PROGRAM F13_CaseContentValidation_ORG
VAR
	fbCrossPushCounter					: CTU;
	bCaseCompleteInsidePacker			: BOOL;


	rtrigSetEarlyCaseValidationOK			: R_TRIG;
	rtrigSetEarlyCaseValidationNOK		: R_TRIG;

	fbBiuldPackerLogString				: FB_CASE_BiuldPackerLogString;
	fbShiftPackerQueue					: FB_CASE_ShiftPackerQueue;
	fbMovePackerToCase				: FB_CASE_MovePackerToCase;
	fbFinaliseCaseData					: FB_CASE_FinaliseCaseData;

	fbValidationIndexOK					: FB_CTU32;
	fbValidationIndexNoData				: FB_CTU32;
	fbValidationIndexUnder				: FB_CTU32;
	fbValidationIndexOver				: FB_CTU32;


	fbDebugCNT				: FB_DEBUG_CounterArray;
	aCNTDebug				: ARRAY [1..10] OF UDINT;
	bResetCNT					: BOOL;


END_VAR

(*
Modification history:
Date		|	Author 		|	Remark
----------------------------------------------------------------------------------------------------
02.09.20	|	PP			|	Start Remarking.
*)

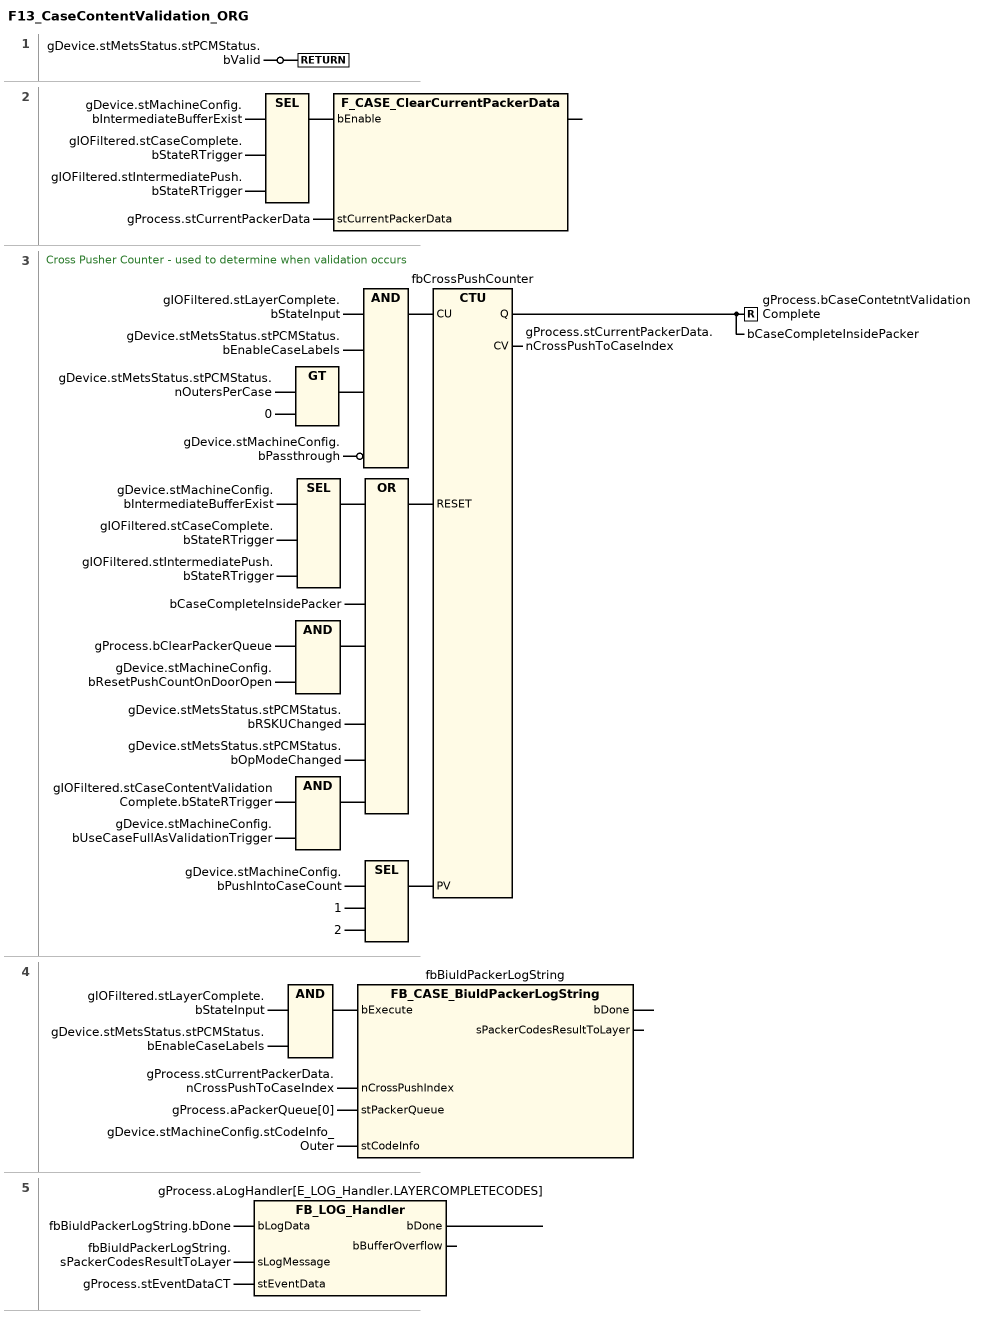
// NETWORK 1
IF NOT gDevice.stMetsStatus.stPCMStatus.bValid THEN RETURN; END_IF

// NETWORK 2
F_CASE_ClearCurrentPackerData(bEnable := SEL(gDevice.stMachineConfig.bIntermediateBufferExist, gIOFiltered.stCaseComplete.bStateRTrigger, gIOFiltered.stIntermediatePush.bStateRTrigger), stCurrentPackerData := gProcess.stCurrentPackerData);

// NETWORK 3
// 					Cross Pusher Counter - used to determine when validation occurs
//
//
fbCrossPushCounter(
    CU := gIOFiltered.stLayerComplete.bStateInput AND gDevice.stMetsStatus.stPCMStatus.bEnableCaseLabels AND gDevice.stMetsStatus.stPCMStatus.nOutersPerCase > 0 AND NOT gDevice.stMachineConfig.bPassthrough,
    RESET := SEL(gDevice.stMachineConfig.bIntermediateBufferExist, gIOFiltered.stCaseComplete.bStateRTrigger, gIOFiltered.stIntermediatePush.bStateRTrigger) OR bCaseCompleteInsidePacker OR gProcess.bClearPackerQueue AND gDevice.stMachineConfig.bResetPushCountOnDoorOpen OR gDevice.stMetsStatus.stPCMStatus.bRSKUChanged OR gDevice.stMetsStatus.stPCMStatus.bOpModeChanged OR gIOFiltered.stCaseContentValidationComplete.bStateRTrigger AND gDevice.stMachineConfig.bUseCaseFullAsValidationTrigger,
    PV := SEL(gDevice.stMachineConfig.bPushIntoCaseCount, 1, 2),
    CV => gProcess.stCurrentPackerData.nCrossPushToCaseIndex); // CTU
gProcess.bCaseContetntValidationComplete R= fbCrossPushCounter.Q;
bCaseCompleteInsidePacker := fbCrossPushCounter.Q;

// NETWORK 4
fbBiuldPackerLogString(
    bExecute := gIOFiltered.stLayerComplete.bStateInput AND gDevice.stMetsStatus.stPCMStatus.bEnableCaseLabels,
    nCrossPushIndex := gProcess.stCurrentPackerData.nCrossPushToCaseIndex,
    stPackerQueue := gProcess.aPackerQueue[0],
    stCodeInfo := gDevice.stMachineConfig.stCodeInfo_Outer); // FB_CASE_BiuldPackerLogString

// NETWORK 5
gProcess.aLogHandler[E_LOG_Handler.LAYERCOMPLETECODES](
    bLogData := fbBiuldPackerLogString.bDone,
    sLogMessage := fbBiuldPackerLogString.sPackerCodesResultToLayer,
    stEventData := gProcess.stEventDataCT); // FB_LOG_Handler

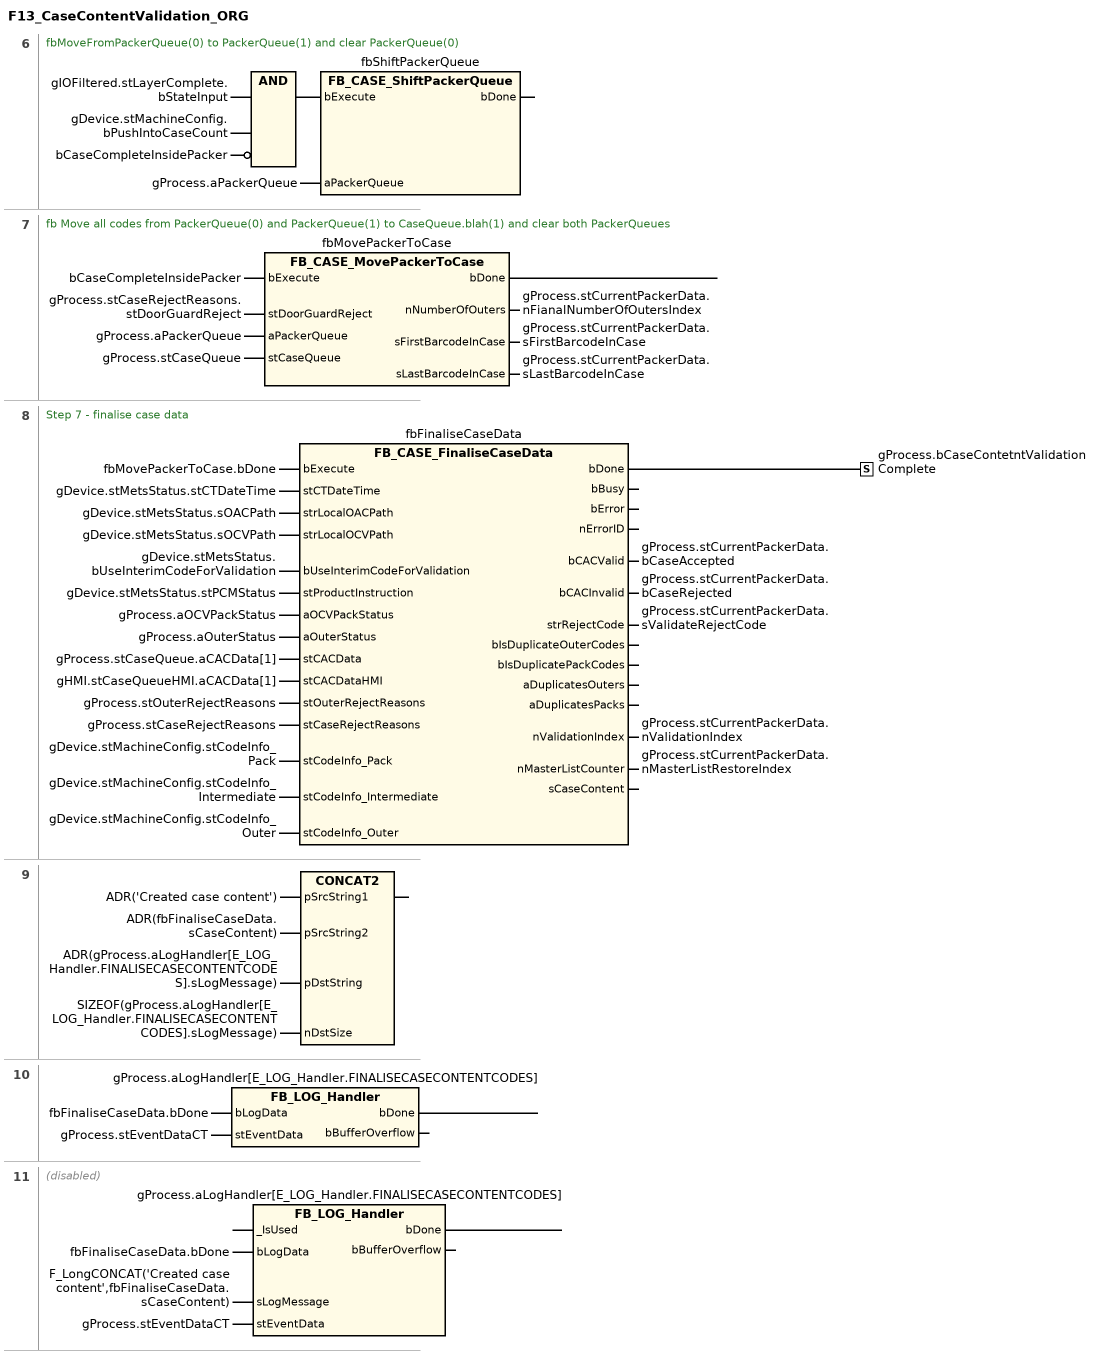
// NETWORK 6
// fbMoveFromPackerQueue(0) to PackerQueue(1) and clear PackerQueue(0)
fbShiftPackerQueue(bExecute := gIOFiltered.stLayerComplete.bStateInput AND gDevice.stMachineConfig.bPushIntoCaseCount AND NOT bCaseCompleteInsidePacker, aPackerQueue := gProcess.aPackerQueue); // FB_CASE_ShiftPackerQueue

// NETWORK 7
// fb Move all codes from PackerQueue(0) and PackerQueue(1) to CaseQueue.blah(1) and clear both PackerQueues
fbMovePackerToCase(
    bExecute := bCaseCompleteInsidePacker,
    stDoorGuardReject := gProcess.stCaseRejectReasons.stDoorGuardReject,
    aPackerQueue := gProcess.aPackerQueue,
    stCaseQueue := gProcess.stCaseQueue,
    nNumberOfOuters => gProcess.stCurrentPackerData.nFianalNumberOfOutersIndex,
    sFirstBarcodeInCase => gProcess.stCurrentPackerData.sFirstBarcodeInCase,
    sLastBarcodeInCase => gProcess.stCurrentPackerData.sLastBarcodeInCase); // FB_CASE_MovePackerToCase

// NETWORK 8
// Step 7 - finalise case data
fbFinaliseCaseData(
    bExecute := fbMovePackerToCase.bDone,
    stCTDateTime := gDevice.stMetsStatus.stCTDateTime,
    strLocalOACPath := gDevice.stMetsStatus.sOACPath,
    strLocalOCVPath := gDevice.stMetsStatus.sOCVPath,
    bUseInterimCodeForValidation := gDevice.stMetsStatus.bUseInterimCodeForValidation,
    stProductInstruction := gDevice.stMetsStatus.stPCMStatus,
    aOCVPackStatus := gProcess.aOCVPackStatus,
    aOuterStatus := gProcess.aOuterStatus,
    stCACData := gProcess.stCaseQueue.aCACData[1],
    stCACDataHMI := gHMI.stCaseQueueHMI.aCACData[1],
    stOuterRejectReasons := gProcess.stOuterRejectReasons,
    stCaseRejectReasons := gProcess.stCaseRejectReasons,
    stCodeInfo_Pack := gDevice.stMachineConfig.stCodeInfo_Pack,
    stCodeInfo_Intermediate := gDevice.stMachineConfig.stCodeInfo_Intermediate,
    stCodeInfo_Outer := gDevice.stMachineConfig.stCodeInfo_Outer,
    bCACValid => gProcess.stCurrentPackerData.bCaseAccepted,
    bCACInvalid => gProcess.stCurrentPackerData.bCaseRejected,
    strRejectCode => gProcess.stCurrentPackerData.sValidateRejectCode,
    nValidationIndex => gProcess.stCurrentPackerData.nValidationIndex,
    nMasterListCounter => gProcess.stCurrentPackerData.nMasterListRestoreIndex); // FB_CASE_FinaliseCaseData
gProcess.bCaseContetntValidationComplete S= fbFinaliseCaseData.bDone;

// NETWORK 9
CONCAT2(pSrcString1 := ADR('Created case content'), pSrcString2 := ADR(fbFinaliseCaseData.sCaseContent), pDstString := ADR(gProcess.aLogHandler[E_LOG_Handler.FINALISECASECONTENTCODES].sLogMessage), nDstSize := SIZEOF(gProcess.aLogHandler[E_LOG_Handler.FINALISECASECONTENTCODES].sLogMessage));

// NETWORK 10
gProcess.aLogHandler[E_LOG_Handler.FINALISECASECONTENTCODES](bLogData := fbFinaliseCaseData.bDone, stEventData := gProcess.stEventDataCT); // FB_LOG_Handler

// NETWORK 11 (disabled)
// gProcess.aLogHandler[E_LOG_Handler.FINALISECASECONTENTCODES](
//     bLogData := fbFinaliseCaseData.bDone,
//     sLogMessage := F_LongCONCAT('Created case content',fbFinaliseCaseData.sCaseContent),
//     stEventData := gProcess.stEventDataCT); // FB_LOG_Handler

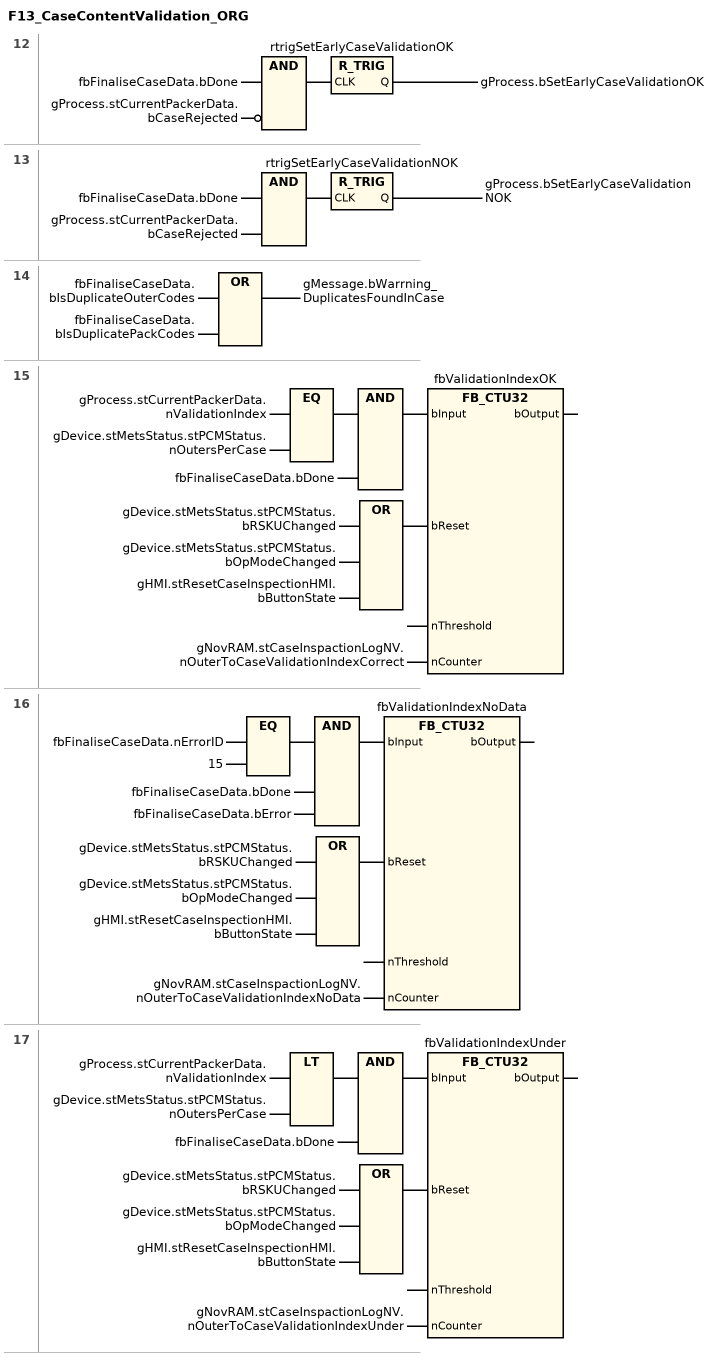
// NETWORK 12
rtrigSetEarlyCaseValidationOK(CLK := fbFinaliseCaseData.bDone AND NOT gProcess.stCurrentPackerData.bCaseRejected); // R_TRIG
gProcess.bSetEarlyCaseValidationOK := rtrigSetEarlyCaseValidationOK.Q;

// NETWORK 13
rtrigSetEarlyCaseValidationNOK(CLK := fbFinaliseCaseData.bDone AND gProcess.stCurrentPackerData.bCaseRejected); // R_TRIG
gProcess.bSetEarlyCaseValidationNOK := rtrigSetEarlyCaseValidationNOK.Q;

// NETWORK 14
gMessage.bWarrning_DuplicatesFoundInCase := fbFinaliseCaseData.bIsDuplicateOuterCodes OR fbFinaliseCaseData.bIsDuplicatePackCodes;

// NETWORK 15
fbValidationIndexOK(
    bInput := gProcess.stCurrentPackerData.nValidationIndex = gDevice.stMetsStatus.stPCMStatus.nOutersPerCase AND fbFinaliseCaseData.bDone,
    bReset := gDevice.stMetsStatus.stPCMStatus.bRSKUChanged OR gDevice.stMetsStatus.stPCMStatus.bOpModeChanged OR gHMI.stResetCaseInspectionHMI.bButtonState,
    nCounter := gNovRAM.stCaseInspactionLogNV.nOuterToCaseValidationIndexCorrect); // FB_CTU32

// NETWORK 16
fbValidationIndexNoData(
    bInput := fbFinaliseCaseData.nErrorID = 15 AND fbFinaliseCaseData.bDone AND fbFinaliseCaseData.bError,
    bReset := gDevice.stMetsStatus.stPCMStatus.bRSKUChanged OR gDevice.stMetsStatus.stPCMStatus.bOpModeChanged OR gHMI.stResetCaseInspectionHMI.bButtonState,
    nCounter := gNovRAM.stCaseInspactionLogNV.nOuterToCaseValidationIndexNoData); // FB_CTU32

// NETWORK 17
fbValidationIndexUnder(
    bInput := gProcess.stCurrentPackerData.nValidationIndex < gDevice.stMetsStatus.stPCMStatus.nOutersPerCase AND fbFinaliseCaseData.bDone,
    bReset := gDevice.stMetsStatus.stPCMStatus.bRSKUChanged OR gDevice.stMetsStatus.stPCMStatus.bOpModeChanged OR gHMI.stResetCaseInspectionHMI.bButtonState,
    nCounter := gNovRAM.stCaseInspactionLogNV.nOuterToCaseValidationIndexUnder); // FB_CTU32

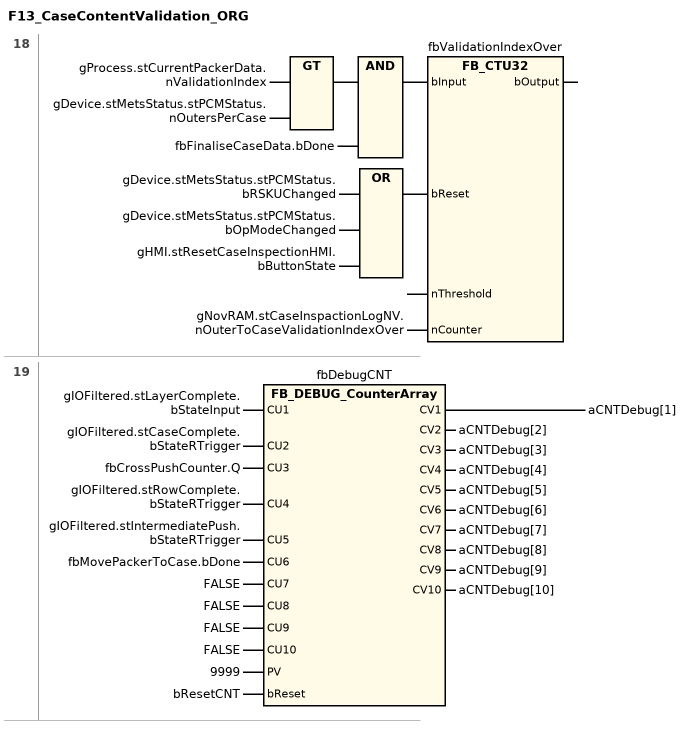
// NETWORK 18
fbValidationIndexOver(
    bInput := gProcess.stCurrentPackerData.nValidationIndex > gDevice.stMetsStatus.stPCMStatus.nOutersPerCase AND fbFinaliseCaseData.bDone,
    bReset := gDevice.stMetsStatus.stPCMStatus.bRSKUChanged OR gDevice.stMetsStatus.stPCMStatus.bOpModeChanged OR gHMI.stResetCaseInspectionHMI.bButtonState,
    nCounter := gNovRAM.stCaseInspactionLogNV.nOuterToCaseValidationIndexOver); // FB_CTU32

// NETWORK 19
fbDebugCNT(
    CU1 := gIOFiltered.stLayerComplete.bStateInput,
    CU2 := gIOFiltered.stCaseComplete.bStateRTrigger,
    CU3 := fbCrossPushCounter.Q,
    CU4 := gIOFiltered.stRowComplete.bStateRTrigger,
    CU5 := gIOFiltered.stIntermediatePush.bStateRTrigger,
    CU6 := fbMovePackerToCase.bDone,
    CU7 := FALSE,
    CU8 := FALSE,
    CU9 := FALSE,
    CU10 := FALSE,
    PV := 9999,
    bReset := bResetCNT,
    CV2 => aCNTDebug[2],
    CV3 => aCNTDebug[3],
    CV4 => aCNTDebug[4],
    CV5 => aCNTDebug[5],
    CV6 => aCNTDebug[6],
    CV7 => aCNTDebug[7],
    CV8 => aCNTDebug[8],
    CV9 => aCNTDebug[9],
    CV10 => aCNTDebug[10]); // FB_DEBUG_CounterArray
aCNTDebug[1] := fbDebugCNT.CV1;

END_PROGRAM

(* stored: Version 1.1.0.1
   POU F13_CaseContentValidation_ORG: Id {72875a2f-e733-400f-92cd-83fb97366fc6}, SpecialFunc None *)
